PROGRAM MAIN
VAR
	Modules: Module_call;
	tAlwaysOn: BOOL; //Temporary BIT FOR Always On
    tAlwaysOff: BOOL; //Temporary BIT FOR Always Off
END_VAR

VAR CONSTANT
END_VAR

// Always ON Logic
tAlwaysOn := TRUE;

// Module call
Modules();

END_PROGRAM

(* stored: Version 1.1.0.1, ProductVersion 3.1.4024.16
   POU MAIN: Id {f4edae46-a55b-4a7f-bfb8-c0711c848216}, SpecialFunc None *)
